// TIA Portal project "move_fieldwrite_read" (V18)

(* hardware
DEVICE "S7-1200 station_1"  S7-1200 Station
   slot 0: "Rack_0"  S7-1200 Rack  Rack  V1.0
   slot 1: "PLC_1"  CPU 1214C DC/DC/DC  6ES7 214-1AG40-0XB0  V4.6
*)

// ===== PLC "PLC_1"  CPU 1214C DC/DC/DC =====

VAR_GLOBAL   // PLC tag table "Default tag table"
   "Tag_1" AT %IB0 : Byte;
   "Tag_2" AT %MD0 : DWord;
   "OKUNAN DEGER" AT %MB10 : Byte;
   "YAZILAN SATIR NO" AT %MD4 : DInt;
END_VAR

DATA_BLOCK "OKUNAN"   // DB1
{ S7_Optimized_Access := 'TRUE' }
VERSION : 0.1
   VAR
      EO : Array[0..10] of Byte;
   END_VAR
BEGIN
   EO[0] := 7;
   EO[1] := 5;
   EO[2] := 1;
   EO[3] := 2;
   EO[4] := 86;
   EO[5] := 14;
   EO[6] := 28;
   EO[7] := 22;
   EO[8] := 11;
   EO[9] := 33;
   EO[10] := 66;
END_DATA_BLOCK

DATA_BLOCK "YAZILAN"   // DB2
{ S7_Optimized_Access := 'TRUE' }
VERSION : 0.1
   VAR
      BBB : Array[0..10] of Byte;
   END_VAR
BEGIN
   BBB[0] := 158;
   BBB[1] := 74;
   BBB[2] := 89;
   BBB[3] := 63;
   BBB[4] := 15;
   BBB[5] := 42;
   BBB[6] := 38;
   BBB[7] := 79;
   BBB[8] := 47;
   BBB[9] := 67;
   BBB[10] := 19;
END_DATA_BLOCK

ORGANIZATION_BLOCK "Main"   // OB1, LAD, ProgramCycle
TITLE = "Main Program Sweep (Cycle)"
{ S7_Optimized_Access := 'TRUE' }
VERSION : 0.1
   VAR_INPUT
      Initial_Call : Bool;   // Initial call of this OB
      Remanence : Bool;   // =True, if remanent data are available
   END_VAR
BEGIN

REGION Network 1
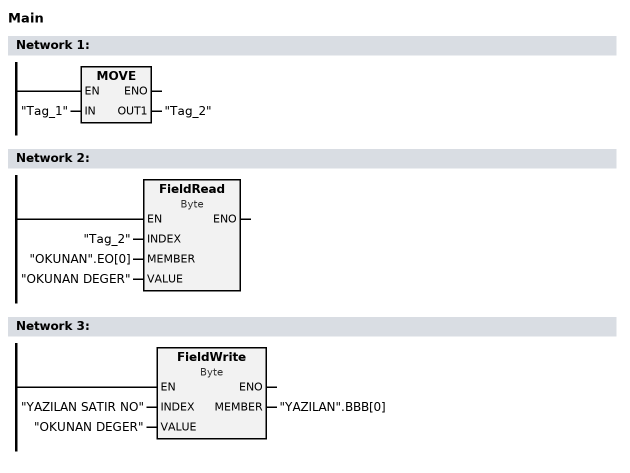
   RUNG wire#powerrail
      Move(in := "Tag_1", out1 => "Tag_2")
   END_RUNG
   // the same network as SCL:
   "Tag_2" := "Tag_1";
END_REGION

REGION Network 2
   // no SCL statement known for FieldRead: written as a call
   FieldRead(index := "Tag_2", member := "OKUNAN".EO[0], value := "OKUNAN DEGER");
END_REGION

REGION Network 3
   // no SCL statement known for FieldWrite: written as a call
   FieldWrite(index := "YAZILAN SATIR NO", value := "OKUNAN DEGER", member => "YAZILAN".BBB[0]);
END_REGION
END_ORGANIZATION_BLOCK